(* IEC 61131-3 sources: DEV_Codegenerator/data/BuR, 4 files *)

(* ---- FB_Std.typ ---- *)
TYPE
TYP_FB_Std : STRUCT
CTRL : FB_Std_CTRL;
STS : FB_Std_STS;
PRM : FB_Std_PRM;
END_STRUCT;

FB_Std_CTRL : STRUCT
Dummy : BOOL; (*Dummy*)
END_STRUCT;

FB_Std_STS : STRUCT
Dummy : BOOL; (*Dummy*)
END_STRUCT;

FB_Std_PRM : STRUCT
Dummy : REAL; (*Dummy*)
END_STRUCT;

END_TYPE

(* ---- FB_Std.fun ---- *)
FUNCTION_BLOCK  FB_Std
VAR_INPUT
IN_Prm_0 : BOOL; (*Input Parameter 1*)
IN_Prm_1 : BOOL; (*Input Parameter 2*)
IN_Prm_2 : BOOL; (*Input Parameter 3*)
IN_Prm_3 : BOOL; (*Input Parameter 4*)
IN_Prm_4 : BOOL; (*Input Parameter 5*)
END_VAR
VAR_OUTPUT
OUT_Prm_0 : BOOL; (*Output Parameter 1*)
OUT_Prm_1 : BOOL; (*Output Parameter 2*)
OUT_Prm_2 : BOOL; (*Output Parameter 3*)
OUT_Prm_3 : BOOL; (*Output Parameter 4*)
OUT_Prm_4 : BOOL; (*Output Parameter 5*)
END_VAR
VAR_IN_OUT
Object_struct : TYP_FB_Std; (*Objectstrucuture*)
END_VAR
END_FUNCTION_BLOCK

(* ---- FB_Std_lib.st ---- *)
//***********************************************
// FB_Std
// Author: dgrill
// Version: 1.0
// Date: 19.12.2018 17:59
// Description:
//
// Interface:
// VAR_INPUT:
// IN_Prm_0:	BOOL	Input Parameter 1
// IN_Prm_1:	BOOL	Input Parameter 2
// IN_Prm_2:	BOOL	Input Parameter 3
// IN_Prm_3:	BOOL	Input Parameter 4
// IN_Prm_4:	BOOL	Input Parameter 5
//
// VAR_OUTPUT:
// OUT_Prm_0:	BOOL	Output Parameter 1
// OUT_Prm_1:	BOOL	Output Parameter 2
// OUT_Prm_2:	BOOL	Output Parameter 3
// OUT_Prm_3:	BOOL	Output Parameter 4
// OUT_Prm_4:	BOOL	Output Parameter 5
//
// VAR_IN_OUT:
// Object_struct:	TYP_FB_Std	Objectstrucuture
//
// Rev:
//
//***********************************************

FUNCTION_BLOCK  FB_Std

// TODO - Insert Code here

END_FUNCTION_BLOCK

(* ---- FB_Std.var ---- *)
VAR
Object1 : FB_Std; (*Standard FB*)
Object2 : FB_Std; (*Standard FB*)
Object3 : FB_Std; (*Standard FB*)
Object4 : FB_Std; (*Standard FB*)
Object5 : FB_Std; (*Standard FB*)
Object6 : FB_Std; (*Standard FB*)
Object7 : FB_Std; (*Standard FB*)
Object8 : FB_Std; (*Standard FB*)
Object9 : FB_Std; (*Standard FB*)
Object10 : FB_Std; (*Standard FB*)
END_VAR
